// TIA Portal V20 export
DATA_BLOCK "InstCallGlobal"   // DB265
// stored: InstanceOfName CallGlobal, InstanceOfType FB
"CallGlobal"
   // VAR
   //    statClockSysMemOld { ExternalWritable := 'False'} : Byte := 16#6B;
   //    statTonTimer : Array[0..1] of IEC_TIMER;
   //    instLAF_PowerOnOff { ExternalWritable := 'False'} : "LAF_PowerOnOff";
   //    instLAF_HmiHeaderManager { ExternalWritable := 'False'} : "LAF_HmiHeaderManager";
   //    instLAF_ClockGen { ExternalWritable := 'False'} : "LAF_ClockGenerator";
   //    instLSNTP_Server { ExternalWritable := 'False'} : "LSNTP_Server";
   //    instRemoteAccess { ExternalWritable := 'False'} : "LRemoteAccess_MobilePanelMonitor";
   //    statPulse : Array[0..99] of Bool;
   // END_VAR
BEGIN
   instLAF_PowerOnOff.on := FALSE;
   instLAF_PowerOnOff.off := FALSE;
   instLAF_PowerOnOff.powerStatus := 0;
   instLAF_PowerOnOff.enablePower := FALSE;
   instLAF_PowerOnOff.statMemOn := FALSE;
   instLAF_HmiHeaderManager.statFirstCall := FALSE;
   instLAF_HmiHeaderManager.statLowerBoundUnit := 0;
   instLAF_HmiHeaderManager.statUpperBoundUnit := 0;
   instLAF_HmiHeaderManager.statLowerBoundHmi := 0;
   instLAF_HmiHeaderManager.statUpperBoundHmi := 1;
   instLAF_HmiHeaderManager.statPreviousSpecialFunction.GaugeRnR1AnodeAlign := FALSE;
   instLAF_HmiHeaderManager.statPreviousSpecialFunction.GaugeRnR1CathodeAlign := FALSE;
   instLAF_HmiHeaderManager.statPreviousSpecialFunction.GaugeRnR3AnodeAlign := FALSE;
   instLAF_HmiHeaderManager.statPreviousSpecialFunction.GaugeRnR3CathodeAlign := FALSE;
   instLAF_HmiHeaderManager.statPreviousSpecialFunction.releaseEntry := FALSE;
   instLAF_HmiHeaderManager.statPreviousSpecialFunction.dryRun := FALSE;
   instLAF_HmiHeaderManager.statPreviousSpecialFunction.RunOut := FALSE;
   instLAF_HmiHeaderManager.statPreviousSpecialFunction.ReworkMode := FALSE;
   instLAF_HmiHeaderManager.statPreviousSpecialFunction.SepaClean := FALSE;
   instLAF_HmiHeaderManager.statPreviousSpecialFunction.MotionUnuse := FALSE;
   instLAF_HmiHeaderManager.statPreviousSpecialFunction.AnodeAlignVisionUnuse := FALSE;
   instLAF_HmiHeaderManager.statPreviousSpecialFunction.CathodeAlignVisionUnuse := FALSE;
   instLAF_HmiHeaderManager.statPreviousSpecialFunction.StackGapVisionUnuse := FALSE;
   instLAF_HmiHeaderManager.statPreviousSpecialFunction.ReelCutAnodeUnuse := FALSE;
   instLAF_HmiHeaderManager.statPreviousSpecialFunction.ReelCutCathodeUnuse := FALSE;
   instLAF_HmiHeaderManager.statPreviousSpecialFunction.InspectionUnuse := FALSE;
   instLAF_ClockGen.clk10Hz := TRUE;
   instLAF_ClockGen.clk5Hz := TRUE;
   instLAF_ClockGen.clk2Hz5 := FALSE;
   instLAF_ClockGen.clk2Hz := TRUE;
   instLAF_ClockGen.clk1Hz25 := FALSE;
   instLAF_ClockGen.clk1Hz := TRUE;
   instLAF_ClockGen.clk0Hz625 := TRUE;
   instLAF_ClockGen.clk0Hz5 := FALSE;
   instLAF_ClockGen.statMemRuntime := 2.78088143015202E-308;
   instLAF_ClockGen.statCalcTimeClk10Hz := 18157;
   instLAF_ClockGen.statCalcTimeClk5Hz := 18157;
   instLAF_ClockGen.statCalcTimeClk2Hz5 := 18157;
   instLAF_ClockGen.statCalcTimeClk2Hz := 18157;
   instLAF_ClockGen.statCalcTimeClk1Hz25 := 218157;
   instLAF_ClockGen.statCalcTimeClk1Hz := 18157;
   instLAF_ClockGen.statCalcTimeClk0Hz625 := 618157;
   instLAF_ClockGen.statCalcTimeClk0Hz5 := 18157;
   instLAF_ClockGen.statStateFlagClk10Hz := FALSE;
   instLAF_ClockGen.statStateFlagClk5Hz := FALSE;
   instLAF_ClockGen.statStateFlagClk2Hz5 := TRUE;
   instLAF_ClockGen.statStateFlagClk2Hz := FALSE;
   instLAF_ClockGen.statStateFlagClk1Hz25 := TRUE;
   instLAF_ClockGen.statStateFlagClk1Hz := FALSE;
   instLAF_ClockGen.statStateFlagClk0Hz625 := FALSE;
   instLAF_ClockGen.statStateFlagClk0Hz5 := TRUE;
   instLSNTP_Server.enable := TRUE;
   instLSNTP_Server.hwID := 64;
   instLSNTP_Server.connID := 16#007B;
   instLSNTP_Server.referenceID := 1;
   instLSNTP_Server.lastTimeSet := DTL#1990-01-01-00:00:00;
   instLSNTP_Server.valid := TRUE;
   instLSNTP_Server.busy := TRUE;
   instLSNTP_Server.error := FALSE;
   instLSNTP_Server.status := 16#7002;
   instLSNTP_Server.diagnostics.status := 16#0000;
   instLSNTP_Server.diagnostics.subfunctionStatus := 16#0000_0000;
   instLSNTP_Server.diagnostics.stateNumber := 0;
   instLSNTP_Server.statEnableOld := TRUE;
   instLSNTP_Server.statValid := TRUE;
   instLSNTP_Server.statBusy := TRUE;
   instLSNTP_Server.statError := FALSE;
   instLSNTP_Server.statErrorUserCleared := FALSE;
   instLSNTP_Server.statErrorAutoCleared := FALSE;
   instLSNTP_Server.statStatus := 16#7002;
   instLSNTP_Server.statSubfunctionStatus := 16#0000;
   instLSNTP_Server.statFBErrorState := 0;
   instLSNTP_Server.statFBState := 50;
   instLSNTP_Server.statDisablingCompleted := FALSE;
   instLSNTP_Server.statEmptyDiagnostics.status := 16#0000;
   instLSNTP_Server.statEmptyDiagnostics.subfunctionStatus := 16#0000_0000;
   instLSNTP_Server.statEmptyDiagnostics.stateNumber := 0;
   instLSNTP_Server.instTCon.REQ := TRUE;
   instLSNTP_Server.instTCon.ID := 16#007B;
   instLSNTP_Server.instTCon.DONE := TRUE;
   instLSNTP_Server.instTCon.BUSY := FALSE;
   instLSNTP_Server.instTCon.ERROR := FALSE;
   instLSNTP_Server.instTCon.STATUS := 16#0000;
   instLSNTP_Server.instTURcv.EN_R := TRUE;
   instLSNTP_Server.instTURcv.ID := 16#007B;
   instLSNTP_Server.instTURcv.LEN := 0;
   instLSNTP_Server.instTURcv.ADHOC := FALSE;
   instLSNTP_Server.instTURcv.NDR := FALSE;
   instLSNTP_Server.instTURcv.BUSY := TRUE;
   instLSNTP_Server.instTURcv.ERROR := FALSE;
   instLSNTP_Server.instTURcv.STATUS := 16#7002;
   instLSNTP_Server.instTURcv.RCVD_LEN := 0;
   instLSNTP_Server.instTUSend.REQ := FALSE;
   instLSNTP_Server.instTUSend.ID := 16#0000;
   instLSNTP_Server.instTUSend.LEN := 0;
   instLSNTP_Server.instTUSend.DONE := FALSE;
   instLSNTP_Server.instTUSend.BUSY := FALSE;
   instLSNTP_Server.instTUSend.ERROR := FALSE;
   instLSNTP_Server.instTUSend.STATUS := 16#7000;
   instLSNTP_Server.instTDiscon.REQ := FALSE;
   instLSNTP_Server.instTDiscon.ID := 16#0000;
   instLSNTP_Server.instTDiscon.DONE := FALSE;
   instLSNTP_Server.instTDiscon.BUSY := FALSE;
   instLSNTP_Server.instTDiscon.ERROR := FALSE;
   instLSNTP_Server.instTDiscon.STATUS := 16#7000;
   instLSNTP_Server.statConParam.InterfaceId := 64;
   instLSNTP_Server.statConParam.ID := 16#007B;
   instLSNTP_Server.statConParam.ConnectionType := 16#13;
   instLSNTP_Server.statConParam.ActiveEstablished := FALSE;
   instLSNTP_Server.statConParam.RemoteAddress.ADDR[1..4] := 16#00;
   instLSNTP_Server.statConParam.RemotePort := 0;
   instLSNTP_Server.statConParam.LocalPort := 123;
   instLSNTP_Server.statAddr.REM_IP_ADDR[1..4] := 0;
   instLSNTP_Server.statAddr.REM_PORT_NR := 0;
   instLSNTP_Server.statAddr.RESERVED := 16#0000;
   instLSNTP_Server.statTelegramRcvd.flags[0..3] := 16#00;
   instLSNTP_Server.statTelegramRcvd.rootDelay := 16#0000_0000;
   instLSNTP_Server.statTelegramRcvd.rootDispersion := 16#0000_0000;
   instLSNTP_Server.statTelegramRcvd.referenceId[0..3] := ' ';
   instLSNTP_Server.statTelegramRcvd.timestamps.reference.sec := 16#0000_0000;
   instLSNTP_Server.statTelegramRcvd.timestamps.reference.secFrac := 16#0000_0000;
   instLSNTP_Server.statTelegramRcvd.timestamps.originate.sec := 16#0000_0000;
   instLSNTP_Server.statTelegramRcvd.timestamps.originate.secFrac := 16#0000_0000;
   instLSNTP_Server.statTelegramRcvd.timestamps.receive.sec := 16#0000_0000;
   instLSNTP_Server.statTelegramRcvd.timestamps.receive.secFrac := 16#0000_0000;
   instLSNTP_Server.statTelegramRcvd.timestamps.transmit.sec := 16#0000_0000;
   instLSNTP_Server.statTelegramRcvd.timestamps.transmit.secFrac := 16#0000_0000;
   instLSNTP_Server.statTelegramRcvd.keyIdentifier := 16#0000_0000;
   instLSNTP_Server.statTelegramRcvd.messageDigest[0..15] := 16#00;
   instLSNTP_Server.statTelegramSend.flags[0..3] := 16#00;
   instLSNTP_Server.statTelegramSend.rootDelay := 16#0000_0000;
   instLSNTP_Server.statTelegramSend.rootDispersion := 16#0000_0000;
   instLSNTP_Server.statTelegramSend.referenceId[0..3] := ' ';
   instLSNTP_Server.statTelegramSend.timestamps.reference.sec := 16#0000_0000;
   instLSNTP_Server.statTelegramSend.timestamps.reference.secFrac := 16#0000_0000;
   instLSNTP_Server.statTelegramSend.timestamps.originate.sec := 16#0000_0000;
   instLSNTP_Server.statTelegramSend.timestamps.originate.secFrac := 16#0000_0000;
   instLSNTP_Server.statTelegramSend.timestamps.receive.sec := 16#0000_0000;
   instLSNTP_Server.statTelegramSend.timestamps.receive.secFrac := 16#0000_0000;
   instLSNTP_Server.statTelegramSend.timestamps.transmit.sec := 16#0000_0000;
   instLSNTP_Server.statTelegramSend.timestamps.transmit.secFrac := 16#0000_0000;
   instLSNTP_Server.statTelegramSend.keyIdentifier := 16#0000_0000;
   instLSNTP_Server.statTelegramSend.messageDigest[0..15] := 16#00;
   instRemoteAccess.lifebitMpPlc := 5;
   instRemoteAccess.connectionTimeOut := T#5S;
   instRemoteAccess.ucpPointerDisabled := FALSE;
   instRemoteAccess.status := 16#0000;
   instRemoteAccess.error := FALSE;
   instRemoteAccess.connectionEnded := FALSE;
   instRemoteAccess.keySwitchMp := 0;
   instRemoteAccess.readoutBoxIdPanel := 0;
   instRemoteAccess.statFirstCall := FALSE;
   instRemoteAccess.statPreviousLifebit := 5;
   instRemoteAccess.statEndConn := FALSE;
   instRemoteAccess.statStatus := 16#0000;
   instRemoteAccess.statLowerBound := 1;
   instRemoteAccess.statUpperBound := 2;
   instRemoteAccess.instTimerLifebit.PT := T#5S;
   instRemoteAccess.instTimerLifebit.IN := TRUE;
END_DATA_BLOCK
